# EPICS substitutions: viocs/si_ps/si_psApp/Db/cs.substitutions
file "db/cs.db" {
    pattern { plane, sector, pos }

        { "H", "01", "M1" }
        { "H", "01", "M2" }
        { "H", "01", "C1-A" }
        { "H", "01", "C1-B" }
        { "H", "01", "C2" }
        { "H", "01", "C4" }
        { "H", "01", "C5-A" }
        { "H", "01", "C5-B" }

        { "V", "01", "M1" }
        { "V", "01", "M2" }
        { "V", "01", "C1" }
        { "V", "01", "C2" }
        { "V", "01", "C4" }
        { "V", "01", "C5" }

        { "H", "02", "M1" }
        { "H", "02", "M2" }
        { "H", "02", "C1-A" }
        { "H", "02", "C1-B" }
        { "H", "02", "C2" }
        { "H", "02", "C4" }
        { "H", "02", "C5-A" }
        { "H", "02", "C5-B" }

        { "V", "02", "M1" }
        { "V", "02", "M2" }
        { "V", "02", "C1" }
        { "V", "02", "C2" }
        { "V", "02", "C4" }
        { "V", "02", "C5" }

        { "H", "03", "M1" }
        { "H", "03", "M2" }
        { "H", "03", "C1-A" }
        { "H", "03", "C1-B" }
        { "H", "03", "C2" }
        { "H", "03", "C4" }
        { "H", "03", "C5-A" }
        { "H", "03", "C5-B" }

        { "V", "03", "M1" }
        { "V", "03", "M2" }
        { "V", "03", "C1" }
        { "V", "03", "C2" }
        { "V", "03", "C4" }
        { "V", "03", "C5" }

        { "H", "04", "M1" }
        { "H", "04", "M2" }
        { "H", "04", "C1-A" }
        { "H", "04", "C1-B" }
        { "H", "04", "C2" }
        { "H", "04", "C4" }
        { "H", "04", "C5-A" }
        { "H", "04", "C5-B" }

        { "V", "04", "M1" }
        { "V", "04", "M2" }
        { "V", "04", "C1" }
        { "V", "04", "C2" }
        { "V", "04", "C4" }
        { "V", "04", "C5" }

        { "H", "05", "M1" }
        { "H", "05", "M2" }
        { "H", "05", "C1-A" }
        { "H", "05", "C1-B" }
        { "H", "05", "C2" }
        { "H", "05", "C4" }
        { "H", "05", "C5-A" }
        { "H", "05", "C5-B" }

        { "V", "05", "M1" }
        { "V", "05", "M2" }
        { "V", "05", "C1" }
        { "V", "05", "C2" }
        { "V", "05", "C4" }
        { "V", "05", "C5" }

        { "H", "06", "M1" }
        { "H", "06", "M2" }
        { "H", "06", "C1-A" }
        { "H", "06", "C1-B" }
        { "H", "06", "C2" }
        { "H", "06", "C4" }
        { "H", "06", "C5-A" }
        { "H", "06", "C5-B" }

        { "V", "06", "M1" }
        { "V", "06", "M2" }
        { "V", "06", "C1" }
        { "V", "06", "C2" }
        { "V", "06", "C4" }
        { "V", "06", "C5" }

        { "H", "07", "M1" }
        { "H", "07", "M2" }
        { "H", "07", "C1-A" }
        { "H", "07", "C1-B" }
        { "H", "07", "C2" }
        { "H", "07", "C4" }
        { "H", "07", "C5-A" }
        { "H", "07", "C5-B" }

        { "V", "07", "M1" }
        { "V", "07", "M2" }
        { "V", "07", "C1" }
        { "V", "07", "C2" }
        { "V", "07", "C4" }
        { "V", "07", "C5" }

        { "H", "08", "M1" }
        { "H", "08", "M2" }
        { "H", "08", "C1-A" }
        { "H", "08", "C1-B" }
        { "H", "08", "C2" }
        { "H", "08", "C4" }
        { "H", "08", "C5-A" }
        { "H", "08", "C5-B" }

        { "V", "08", "M1" }
        { "V", "08", "M2" }
        { "V", "08", "C1" }
        { "V", "08", "C2" }
        { "V", "08", "C4" }
        { "V", "08", "C5" }

        { "H", "09", "M1" }
        { "H", "09", "M2" }
        { "H", "09", "C1-A" }
        { "H", "09", "C1-B" }
        { "H", "09", "C2" }
        { "H", "09", "C4" }
        { "H", "09", "C5-A" }
        { "H", "09", "C5-B" }

        { "V", "09", "M1" }
        { "V", "09", "M2" }
        { "V", "09", "C1" }
        { "V", "09", "C2" }
        { "V", "09", "C4" }
        { "V", "09", "C5" }

        { "H", "10", "M1" }
        { "H", "10", "M2" }
        { "H", "10", "C1-A" }
        { "H", "10", "C1-B" }
        { "H", "10", "C2" }
        { "H", "10", "C4" }
        { "H", "10", "C5-A" }
        { "H", "10", "C5-B" }

        { "V", "10", "M1" }
        { "V", "10", "M2" }
        { "V", "10", "C1" }
        { "V", "10", "C2" }
        { "V", "10", "C4" }
        { "V", "10", "C5" }

        { "H", "11", "M1" }
        { "H", "11", "M2" }
        { "H", "11", "C1-A" }
        { "H", "11", "C1-B" }
        { "H", "11", "C2" }
        { "H", "11", "C4" }
        { "H", "11", "C5-A" }
        { "H", "11", "C5-B" }

        { "V", "11", "M1" }
        { "V", "11", "M2" }
        { "V", "11", "C1" }
        { "V", "11", "C2" }
        { "V", "11", "C4" }
        { "V", "11", "C5" }

        { "H", "12", "M1" }
        { "H", "12", "M2" }
        { "H", "12", "C1-A" }
        { "H", "12", "C1-B" }
        { "H", "12", "C2" }
        { "H", "12", "C4" }
        { "H", "12", "C5-A" }
        { "H", "12", "C5-B" }

        { "V", "12", "M1" }
        { "V", "12", "M2" }
        { "V", "12", "C1" }
        { "V", "12", "C2" }
        { "V", "12", "C4" }
        { "V", "12", "C5" }

        { "H", "13", "M1" }
        { "H", "13", "M2" }
        { "H", "13", "C1-A" }
        { "H", "13", "C1-B" }
        { "H", "13", "C2" }
        { "H", "13", "C4" }
        { "H", "13", "C5-A" }
        { "H", "13", "C5-B" }

        { "V", "13", "M1" }
        { "V", "13", "M2" }
        { "V", "13", "C1" }
        { "V", "13", "C2" }
        { "V", "13", "C4" }
        { "V", "13", "C5" }

        { "H", "14", "M1" }
        { "H", "14", "M2" }
        { "H", "14", "C1-A" }
        { "H", "14", "C1-B" }
        { "H", "14", "C2" }
        { "H", "14", "C4" }
        { "H", "14", "C5-A" }
        { "H", "14", "C5-B" }

        { "V", "14", "M1" }
        { "V", "14", "M2" }
        { "V", "14", "C1" }
        { "V", "14", "C2" }
        { "V", "14", "C4" }
        { "V", "14", "C5" }

        { "H", "15", "M1" }
        { "H", "15", "M2" }
        { "H", "15", "C1-A" }
        { "H", "15", "C1-B" }
        { "H", "15", "C2" }
        { "H", "15", "C4" }
        { "H", "15", "C5-A" }
        { "H", "15", "C5-B" }

        { "V", "15", "M1" }
        { "V", "15", "M2" }
        { "V", "15", "C1" }
        { "V", "15", "C2" }
        { "V", "15", "C4" }
        { "V", "15", "C5" }

        { "H", "16", "M1" }
        { "H", "16", "M2" }
        { "H", "16", "C1-A" }
        { "H", "16", "C1-B" }
        { "H", "16", "C2" }
        { "H", "16", "C4" }
        { "H", "16", "C5-A" }
        { "H", "16", "C5-B" }

        { "V", "16", "M1" }
        { "V", "16", "M2" }
        { "V", "16", "C1" }
        { "V", "16", "C2" }
        { "V", "16", "C4" }
        { "V", "16", "C5" }

        { "H", "17", "M1" }
        { "H", "17", "M2" }
        { "H", "17", "C1-A" }
        { "H", "17", "C1-B" }
        { "H", "17", "C2" }
        { "H", "17", "C4" }
        { "H", "17", "C5-A" }
        { "H", "17", "C5-B" }

        { "V", "17", "M1" }
        { "V", "17", "M2" }
        { "V", "17", "C1" }
        { "V", "17", "C2" }
        { "V", "17", "C4" }
        { "V", "17", "C5" }

        { "H", "18", "M1" }
        { "H", "18", "M2" }
        { "H", "18", "C1-A" }
        { "H", "18", "C1-B" }
        { "H", "18", "C2" }
        { "H", "18", "C4" }
        { "H", "18", "C5-A" }
        { "H", "18", "C5-B" }

        { "V", "18", "M1" }
        { "V", "18", "M2" }
        { "V", "18", "C1" }
        { "V", "18", "C2" }
        { "V", "18", "C4" }
        { "V", "18", "C5" }

        { "H", "19", "M1" }
        { "H", "19", "M2" }
        { "H", "19", "C1-A" }
        { "H", "19", "C1-B" }
        { "H", "19", "C2" }
        { "H", "19", "C4" }
        { "H", "19", "C5-A" }
        { "H", "19", "C5-B" }

        { "V", "19", "M1" }
        { "V", "19", "M2" }
        { "V", "19", "C1" }
        { "V", "19", "C2" }
        { "V", "19", "C4" }
        { "V", "19", "C5" }

        { "H", "20", "M1" }
        { "H", "20", "M2" }
        { "H", "20", "C1-A" }
        { "H", "20", "C1-B" }
        { "H", "20", "C2" }
        { "H", "20", "C4" }
        { "H", "20", "C5-A" }
        { "H", "20", "C5-B" }

        { "V", "20", "M1" }
        { "V", "20", "M2" }
        { "V", "20", "C1" }
        { "V", "20", "C2" }
        { "V", "20", "C4" }
        { "V", "20", "C5" }

}
